// Block: Area03_Messages

DATA_BLOCK Area03_Messages
VERSION : 0.1
   NON_RETAIN
   VAR
      A : Struct
         Msg : Array[1..736] of Bool;
         Hmi : Array[1..46] of Word;
         Ack : Array[1..46] of Word;
      END_STRUCT;
      W : Struct
         Msg : Array[1..832] of Bool;
         Hmi : Array[1..52] of Word;
         Ack : Array[1..52] of Word;
      END_STRUCT;
   END_VAR

BEGIN
   // No initialization required
END_DATA_BLOCK
